FUNCTION_BLOCK Stopping IMPLEMENTS ITF_PackMLState
VAR
END_VAR

METHOD CyclicLogic : BOOL
VAR_INPUT
END_VAR
END_METHOD

{warning 'add method implementation '}
METHOD EStop : BOOL
END_METHOD

{warning 'add method implementation '}
METHOD Reset : BOOL
END_METHOD

{warning 'add method implementation '}
METHOD Start : BOOL
END_METHOD

{warning 'add method implementation '}
METHOD Stop : BOOL
END_METHOD

END_FUNCTION_BLOCK

(* stored: Version 1.1.0.1, ProductVersion 3.1.4024.12
   POU Stopping: Id {9157fb53-3b36-484b-96f5-31503e53a781}, SpecialFunc None
   Method CyclicLogic: Id {b1c4d5e0-f2e7-46dc-be85-09efde05b463}
   Method EStop: Id {46f7e2a4-ecb5-4195-a804-c9cbc0ab0701}
   Method Reset: Id {d53d2e7b-fd5f-4594-bc83-6f2da0e134a4}
   Method Start: Id {1f2401c8-e5f5-4847-8e73-edd8f35c4748}
   Method Stop: Id {a881fa75-46f2-4c5d-8fcc-f63f6f6316fc} *)
